FUNCTION TryConvert_USINT_TO_BYTE : BOOL
VAR_INPUT
	in : USINT;
	out : REFERENCE TO BYTE;
END_VAR

out := USINT_TO_BYTE(in);
TryConvert_USINT_TO_BYTE := TRUE;

END_FUNCTION

(* stored: Version 1.1.0.1, ProductVersion 3.1.4024.12
   POU TryConvert_USINT_TO_BYTE: Id {5fcdea9c-e20c-48a7-8913-1c8b44fd8d3b}, SpecialFunc None *)
